# EPICS autosave request: iocBoot/iocAndor3/auto_settings.req
file "ADBase_settings.req",       P=$(P),  R=cam1:
#file "andor3_settings.req",       P=$(P),  R=cam1:
#file "NDFile_settings.req",       P=$(P),  R=cam1:
file "NDPluginBase_settings.req", P=$(P),  R=image1:
file "NDStdArrays_settings.req",  P=$(P),  R=image1:
file "commonPlugin_settings.req", P=$(P)
